Fanuc KAREL source: RENAME_FILE.kl

PROGRAM T
%NOLOCKGROUP
VAR
 v0 : STRING[40]
 v1 : STRING[40]
 v2 : BOOLEAN
 v3 : INTEGER
BEGIN
 RENAME_FILE(v0, v1, v2, v3)
END T
